Omron CX-Programmer project NewProject (CX-Programmer 9.75)

# PLC Learning: CJ2M CPU11

## Program NewProgram1 (cyclic task 0)
Local symbols
FM 100.01 BOOL
Lamp2 100.04 BOOL
M 100.00 BOOL
RM 100.03 BOOL
Sw1 0.00 BOOL
Sw2 0.01 BOOL
Sw3 0.02 BOOL
Sw5 0.04 BOOL
Sw6 0.05 BOOL
lamp1 100.02 BOOL
sw4 0.03 BOOL

### Section Section1

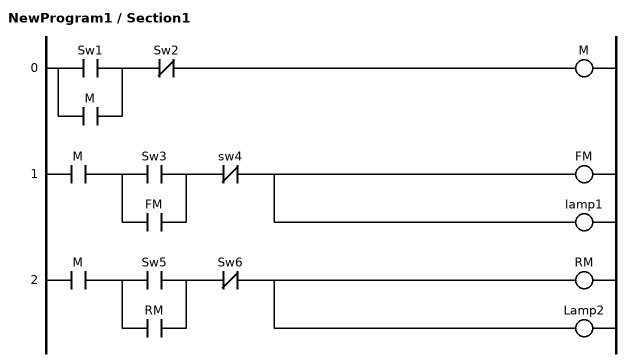
; rung 0
LD Sw1
OR M
ANDNOT Sw2
OUT M
; rung 1
LD M
LD Sw3
OR FM
ANDLD
ANDNOT sw4
OUT FM
OUT lamp1
; rung 2
LD M
LD Sw5
OR RM
ANDLD
ANDNOT Sw6
OUT RM
OUT Lamp2

### Section END
; rung 0
END(001)